VAR_GLOBAL
	fbConfiguration		: FB_Configuration;
	fbObjectDirectory 	: FB_ObjectDirectory;
	nObjPropChangeCnt	: USINT;
END_VAR

(* stored: Version 1.1.0.1, ProductVersion 3.1.4022.12
   GVL GVL_ObjMgmt: Id {539d25b4-2a96-45e3-bd06-1ea86955fb48} *)
